// TIA Portal V20 export
VAR_GLOBAL   // PLC tag table "Cabinet14"
   Sz14_Column_Buzzer AT %Q1201.5 : Bool;
   Sz14_Column_Red AT %Q1201.3 : Bool;
   Sz14_Column_Yellow AT %Q1201.1 : Bool;
   Sz14_Column_Green AT %Q1200.7 : Bool;
END_VAR
